// TIA Portal V21 export
FUNCTION "ALARMS" : Void   // FC8, LAD
{ S7_Optimized_Access := 'TRUE' }
// stored: SetENOAutomatically false
   VAR_TEMP   // added for the SCL form of the ladder/FBD networks
      _w1 : Bool;
      _w2 : Bool;
      _w3 : Bool;
      _w4 : Bool;
   END_VAR
BEGIN

REGION Network 1: ERROR
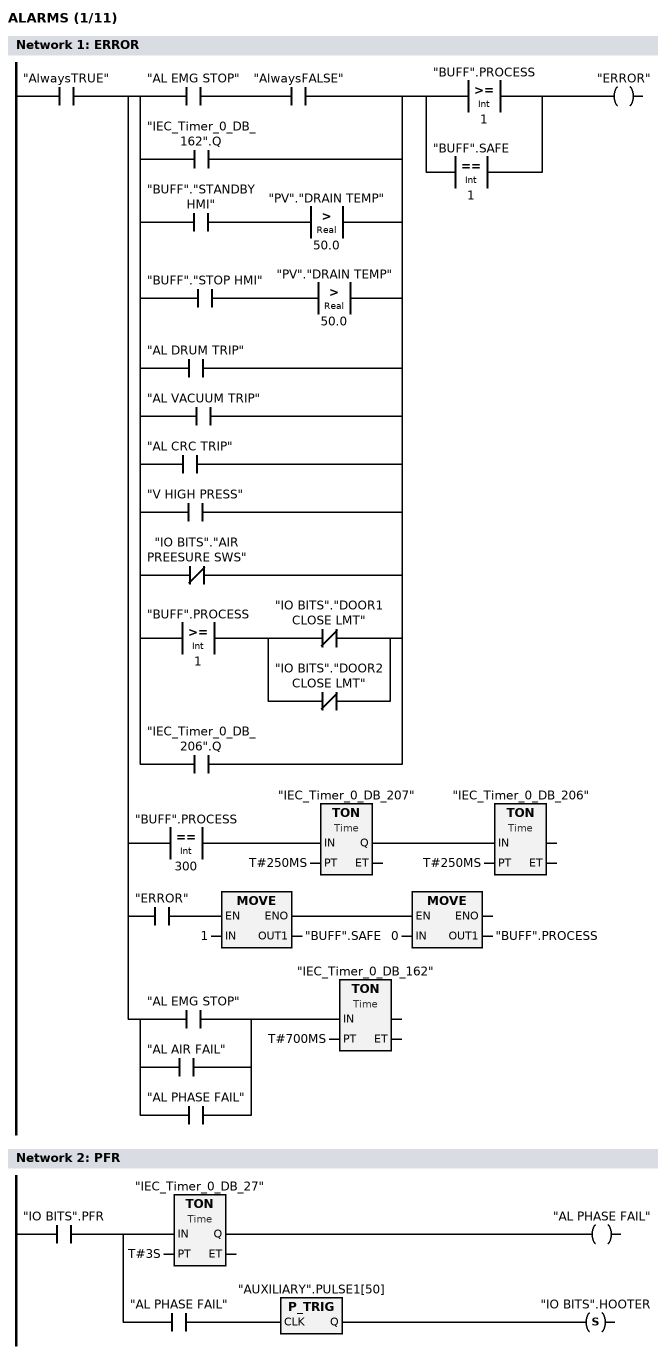
   RUNG wire#powerrail
      Contact( "AlwaysTRUE" )
      wire#w1
      Contact( "AL EMG STOP" )
      Contact( "AlwaysFALSE" )
      wire#w2
      { S7_Templates := "SrcType := Int" } GE_Contact(in1 := "BUFF".PROCESS, in2 := 1)
      wire#w4
      Coil( "ERROR" )
   END_RUNG
   RUNG wire#w1
      Contact( "IEC_Timer_0_DB_162".Q )
   END_RUNG wire#w2
   RUNG wire#w1
      Contact( "BUFF"."STANDBY HMI" )
      { S7_Templates := "SrcType := Real" } GT_Contact(in1 := "PV"."DRAIN TEMP", in2 := 50.0)
   END_RUNG wire#w2
   RUNG wire#w1
      Contact( "BUFF"."STOP HMI" )
      { S7_Templates := "SrcType := Real" } GT_Contact(in1 := "PV"."DRAIN TEMP", in2 := 50.0)
   END_RUNG wire#w2
   RUNG wire#w1
      Contact( "AL DRUM TRIP" )
   END_RUNG wire#w2
   RUNG wire#w1
      Contact( "AL VACUUM TRIP" )
   END_RUNG wire#w2
   RUNG wire#w1
      Contact( "AL CRC TRIP" )
   END_RUNG wire#w2
   RUNG wire#w1
      Contact( "V HIGH PRESS" )
   END_RUNG wire#w2
   RUNG wire#w1
      I_Contact( "IO BITS"."AIR PREESURE SWS" )
   END_RUNG wire#w2
   RUNG wire#w1
      { S7_Templates := "SrcType := Int" } GE_Contact(in1 := "BUFF".PROCESS, in2 := 1)
      wire#w3
      I_Contact( "IO BITS"."DOOR1 CLOSE LMT" )
   END_RUNG wire#w2
   RUNG wire#w3
      I_Contact( "IO BITS"."DOOR2 CLOSE LMT" )
   END_RUNG wire#w2
   RUNG wire#w1
      Contact( "IEC_Timer_0_DB_206".Q )
   END_RUNG wire#w2
   RUNG wire#w2
      { S7_Templates := "SrcType := Int" } EQ_Contact(in1 := "BUFF".SAFE, in2 := 1)
   END_RUNG wire#w4
   RUNG wire#w1
      { S7_Templates := "SrcType := Int" } EQ_Contact(in1 := "BUFF".PROCESS, in2 := 300)
      { S7_Templates := "time_type := Time" } "IEC_Timer_0_DB_207".TON(pt := T#250MS, et =>)
      { S7_Templates := "time_type := Time" } "IEC_Timer_0_DB_206".TON(pt := T#250MS, et =>)
   END_RUNG
   RUNG wire#w1
      Contact( "ERROR" )
      Move(in := 1, out1 => "BUFF".SAFE)
      Move(in := 0, out1 => "BUFF".PROCESS)
   END_RUNG
   RUNG wire#w1
      Contact( "AL EMG STOP" )
      wire#w5
      { S7_Templates := "time_type := Time" } "IEC_Timer_0_DB_162".TON(pt := T#700MS, et =>)
   END_RUNG
   RUNG wire#w1
      Contact( "AL AIR FAIL" )
   END_RUNG wire#w5
   RUNG wire#w1
      Contact( "AL PHASE FAIL" )
   END_RUNG wire#w5
   // the same network as SCL:
   "ERROR" := "AlwaysTRUE" AND (("AL EMG STOP" AND "AlwaysFALSE") OR "IEC_Timer_0_DB_162".Q OR ("BUFF"."STANDBY HMI" AND ("PV"."DRAIN TEMP" > 50.0)) OR ("BUFF"."STOP HMI" AND ("PV"."DRAIN TEMP" > 50.0)) OR "AL DRUM TRIP" OR "AL VACUUM TRIP" OR "AL CRC TRIP" OR "V HIGH PRESS" OR NOT "IO BITS"."AIR PREESURE SWS" OR (("BUFF".PROCESS >= 1) AND (NOT "IO BITS"."DOOR1 CLOSE LMT" OR NOT "IO BITS"."DOOR2 CLOSE LMT")) OR "IEC_Timer_0_DB_206".Q) AND (("BUFF".PROCESS >= 1) OR ("BUFF".SAFE = 1));
   "IEC_Timer_0_DB_207".TON(IN := "AlwaysTRUE" AND ("BUFF".PROCESS = 300), PT := T#250MS);
   "IEC_Timer_0_DB_206".TON(IN := "IEC_Timer_0_DB_207".Q, PT := T#250MS);
   IF "AlwaysTRUE" AND "ERROR" THEN
       "BUFF".SAFE := 1;
       "BUFF".PROCESS := 0;
   END_IF;
   "IEC_Timer_0_DB_162".TON(IN := "AlwaysTRUE" AND ("AL EMG STOP" OR "AL AIR FAIL" OR "AL PHASE FAIL"),
                           PT := T#700MS);
END_REGION

REGION Network 2: PFR
   RUNG wire#powerrail
      Contact( "IO BITS".PFR )
      wire#w1
      { S7_Templates := "time_type := Time" } "IEC_Timer_0_DB_27".TON(pt := T#3S, et =>)
      Coil( "AL PHASE FAIL" )
   END_RUNG
   RUNG wire#w1
      Contact( "AL PHASE FAIL" )
      P_Trig( "AUXILIARY".PULSE1[50] )
      S_Coil( "IO BITS".HOOTER )
   END_RUNG
   // the same network as SCL:
   "IEC_Timer_0_DB_27".TON(IN := "IO BITS".PFR, PT := T#3S);
   "AL PHASE FAIL" := "IEC_Timer_0_DB_27".Q;
   #_w1 := "IO BITS".PFR AND "AL PHASE FAIL";
   #_w2 := #_w1 AND NOT "AUXILIARY".PULSE1[50];   // rising edge
   "AUXILIARY".PULSE1[50] := #_w1;
   IF #_w2 THEN "IO BITS".HOOTER := TRUE; END_IF;
END_REGION

REGION Network 3: EMG
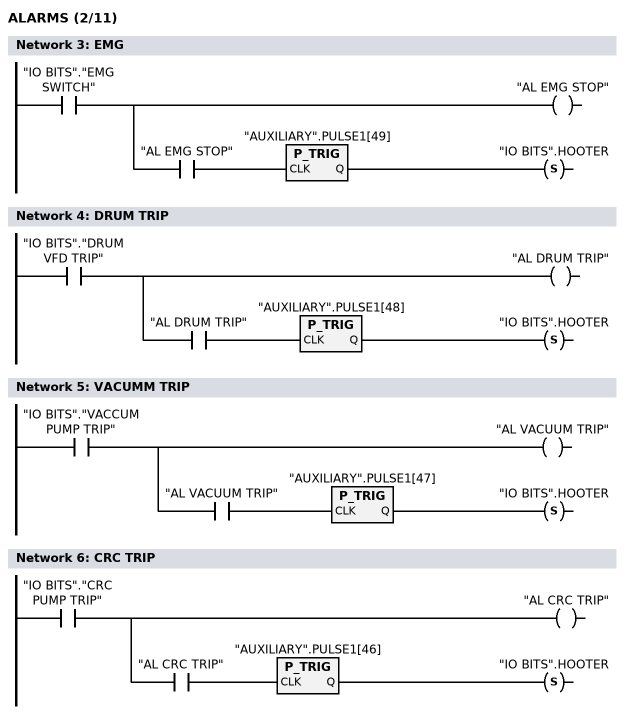
   RUNG wire#powerrail
      Contact( "IO BITS"."EMG SWITCH" )
      wire#w1
      Coil( "AL EMG STOP" )
   END_RUNG
   RUNG wire#w1
      Contact( "AL EMG STOP" )
      P_Trig( "AUXILIARY".PULSE1[49] )
      S_Coil( "IO BITS".HOOTER )
   END_RUNG
   // the same network as SCL:
   "AL EMG STOP" := "IO BITS"."EMG SWITCH";
   #_w1 := "IO BITS"."EMG SWITCH" AND "AL EMG STOP";
   #_w2 := #_w1 AND NOT "AUXILIARY".PULSE1[49];   // rising edge
   "AUXILIARY".PULSE1[49] := #_w1;
   IF #_w2 THEN "IO BITS".HOOTER := TRUE; END_IF;
END_REGION

REGION Network 4: DRUM TRIP
   RUNG wire#powerrail
      Contact( "IO BITS"."DRUM VFD TRIP" )
      wire#w1
      Coil( "AL DRUM TRIP" )
   END_RUNG
   RUNG wire#w1
      Contact( "AL DRUM TRIP" )
      P_Trig( "AUXILIARY".PULSE1[48] )
      S_Coil( "IO BITS".HOOTER )
   END_RUNG
   // the same network as SCL:
   "AL DRUM TRIP" := "IO BITS"."DRUM VFD TRIP";
   #_w1 := "IO BITS"."DRUM VFD TRIP" AND "AL DRUM TRIP";
   #_w2 := #_w1 AND NOT "AUXILIARY".PULSE1[48];   // rising edge
   "AUXILIARY".PULSE1[48] := #_w1;
   IF #_w2 THEN "IO BITS".HOOTER := TRUE; END_IF;
END_REGION

REGION Network 5: VACUMM TRIP
   RUNG wire#powerrail
      Contact( "IO BITS"."VACCUM PUMP TRIP" )
      wire#w1
      Coil( "AL VACUUM TRIP" )
   END_RUNG
   RUNG wire#w1
      Contact( "AL VACUUM TRIP" )
      P_Trig( "AUXILIARY".PULSE1[47] )
      S_Coil( "IO BITS".HOOTER )
   END_RUNG
   // the same network as SCL:
   "AL VACUUM TRIP" := "IO BITS"."VACCUM PUMP TRIP";
   #_w1 := "IO BITS"."VACCUM PUMP TRIP" AND "AL VACUUM TRIP";
   #_w2 := #_w1 AND NOT "AUXILIARY".PULSE1[47];   // rising edge
   "AUXILIARY".PULSE1[47] := #_w1;
   IF #_w2 THEN "IO BITS".HOOTER := TRUE; END_IF;
END_REGION

REGION Network 6: CRC TRIP
   RUNG wire#powerrail
      Contact( "IO BITS"."CRC PUMP TRIP" )
      wire#w1
      Coil( "AL CRC TRIP" )
   END_RUNG
   RUNG wire#w1
      Contact( "AL CRC TRIP" )
      P_Trig( "AUXILIARY".PULSE1[46] )
      S_Coil( "IO BITS".HOOTER )
   END_RUNG
   // the same network as SCL:
   "AL CRC TRIP" := "IO BITS"."CRC PUMP TRIP";
   #_w1 := "IO BITS"."CRC PUMP TRIP" AND "AL CRC TRIP";
   #_w2 := #_w1 AND NOT "AUXILIARY".PULSE1[46];   // rising edge
   "AUXILIARY".PULSE1[46] := #_w1;
   IF #_w2 THEN "IO BITS".HOOTER := TRUE; END_IF;
END_REGION

REGION Network 7: PROCESS START AND OVER
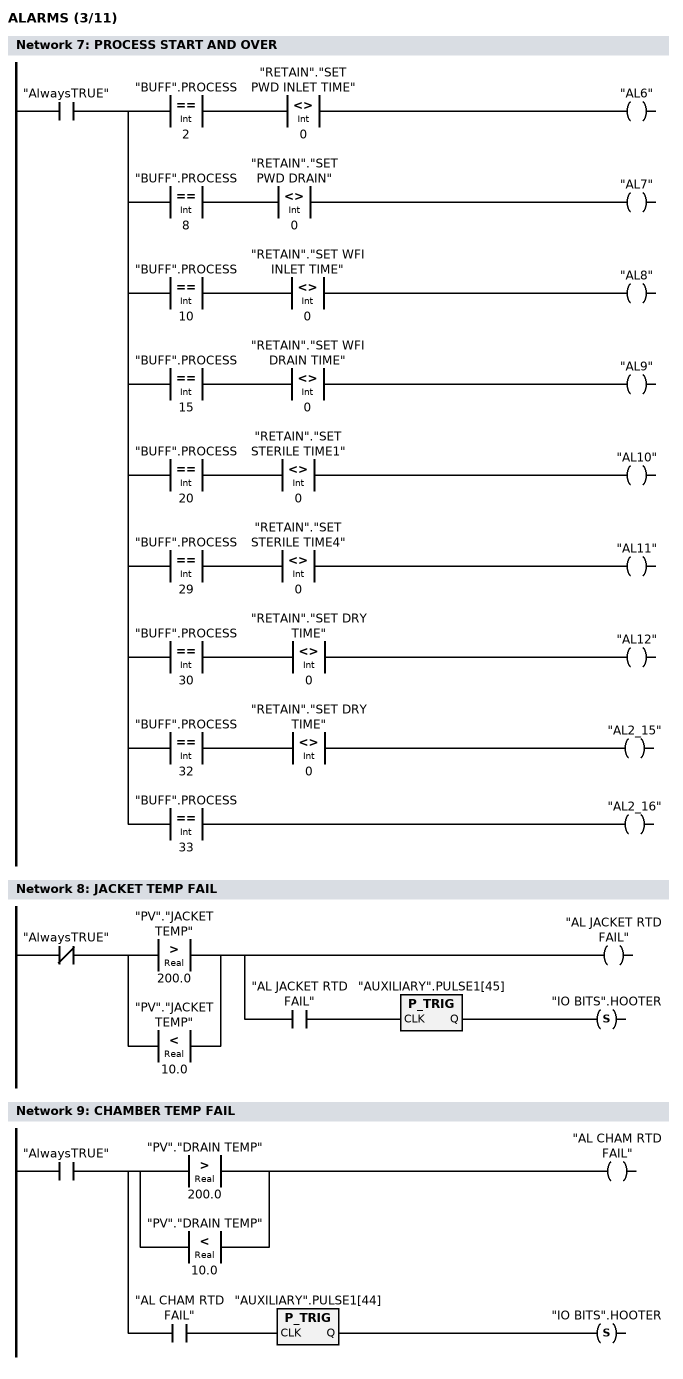
   RUNG wire#powerrail
      Contact( "AlwaysTRUE" )
      wire#w1
      { S7_Templates := "SrcType := Int" } EQ_Contact(in1 := "BUFF".PROCESS, in2 := 2)
      { S7_Templates := "SrcType := Int" } NE_Contact(in1 := "RETAIN"."SET PWD INLET TIME", in2 := 0)
      Coil( "AL6" )
   END_RUNG
   RUNG wire#w1
      { S7_Templates := "SrcType := Int" } EQ_Contact(in1 := "BUFF".PROCESS, in2 := 8)
      { S7_Templates := "SrcType := Int" } NE_Contact(in1 := "RETAIN"."SET PWD DRAIN", in2 := 0)
      Coil( "AL7" )
   END_RUNG
   RUNG wire#w1
      { S7_Templates := "SrcType := Int" } EQ_Contact(in1 := "BUFF".PROCESS, in2 := 10)
      { S7_Templates := "SrcType := Int" } NE_Contact(in1 := "RETAIN"."SET WFI INLET TIME", in2 := 0)
      Coil( "AL8" )
   END_RUNG
   RUNG wire#w1
      { S7_Templates := "SrcType := Int" } EQ_Contact(in1 := "BUFF".PROCESS, in2 := 15)
      { S7_Templates := "SrcType := Int" } NE_Contact(in1 := "RETAIN"."SET WFI DRAIN TIME", in2 := 0)
      Coil( "AL9" )
   END_RUNG
   RUNG wire#w1
      { S7_Templates := "SrcType := Int" } EQ_Contact(in1 := "BUFF".PROCESS, in2 := 20)
      { S7_Templates := "SrcType := Int" } NE_Contact(in1 := "RETAIN"."SET STERILE TIME1", in2 := 0)
      Coil( "AL10" )
   END_RUNG
   RUNG wire#w1
      { S7_Templates := "SrcType := Int" } EQ_Contact(in1 := "BUFF".PROCESS, in2 := 29)
      { S7_Templates := "SrcType := Int" } NE_Contact(in1 := "RETAIN"."SET STERILE TIME4", in2 := 0)
      Coil( "AL11" )
   END_RUNG
   RUNG wire#w1
      { S7_Templates := "SrcType := Int" } EQ_Contact(in1 := "BUFF".PROCESS, in2 := 30)
      { S7_Templates := "SrcType := Int" } NE_Contact(in1 := "RETAIN"."SET DRY TIME", in2 := 0)
      Coil( "AL12" )
   END_RUNG
   RUNG wire#w1
      { S7_Templates := "SrcType := Int" } EQ_Contact(in1 := "BUFF".PROCESS, in2 := 32)
      { S7_Templates := "SrcType := Int" } NE_Contact(in1 := "RETAIN"."SET DRY TIME", in2 := 0)
      Coil( "AL2_15" )
   END_RUNG
   RUNG wire#w1
      { S7_Templates := "SrcType := Int" } EQ_Contact(in1 := "BUFF".PROCESS, in2 := 33)
      Coil( "AL2_16" )
   END_RUNG
   // the same network as SCL:
   "AL6" := "AlwaysTRUE" AND ("BUFF".PROCESS = 2) AND ("RETAIN"."SET PWD INLET TIME" <> 0);
   "AL7" := "AlwaysTRUE" AND ("BUFF".PROCESS = 8) AND ("RETAIN"."SET PWD DRAIN" <> 0);
   "AL8" := "AlwaysTRUE" AND ("BUFF".PROCESS = 10) AND ("RETAIN"."SET WFI INLET TIME" <> 0);
   "AL9" := "AlwaysTRUE" AND ("BUFF".PROCESS = 15) AND ("RETAIN"."SET WFI DRAIN TIME" <> 0);
   "AL10" := "AlwaysTRUE" AND ("BUFF".PROCESS = 20) AND ("RETAIN"."SET STERILE TIME1" <> 0);
   "AL11" := "AlwaysTRUE" AND ("BUFF".PROCESS = 29) AND ("RETAIN"."SET STERILE TIME4" <> 0);
   "AL12" := "AlwaysTRUE" AND ("BUFF".PROCESS = 30) AND ("RETAIN"."SET DRY TIME" <> 0);
   "AL2_15" := "AlwaysTRUE" AND ("BUFF".PROCESS = 32) AND ("RETAIN"."SET DRY TIME" <> 0);
   "AL2_16" := "AlwaysTRUE" AND ("BUFF".PROCESS = 33);
END_REGION

REGION Network 8: JACKET TEMP FAIL
   RUNG wire#powerrail
      I_Contact( "AlwaysTRUE" )
      wire#w1
      { S7_Templates := "SrcType := Real" } GT_Contact(in1 := "PV"."JACKET TEMP", in2 := 200.0)
      wire#w2
      Coil( "AL JACKET RTD FAIL" )
   END_RUNG
   RUNG wire#w1
      { S7_Templates := "SrcType := Real" } LT_Contact(in1 := "PV"."JACKET TEMP", in2 := 10.0)
   END_RUNG wire#w2
   RUNG wire#w2
      Contact( "AL JACKET RTD FAIL" )
      P_Trig( "AUXILIARY".PULSE1[45] )
      S_Coil( "IO BITS".HOOTER )
   END_RUNG
   // the same network as SCL:
   "AL JACKET RTD FAIL" := NOT "AlwaysTRUE" AND (("PV"."JACKET TEMP" > 200.0) OR ("PV"."JACKET TEMP" < 10.0));
   #_w1 := "AL JACKET RTD FAIL" AND "AL JACKET RTD FAIL";
   #_w2 := #_w1 AND NOT "AUXILIARY".PULSE1[45];   // rising edge
   "AUXILIARY".PULSE1[45] := #_w1;
   IF #_w2 THEN "IO BITS".HOOTER := TRUE; END_IF;
END_REGION

REGION Network 9: CHAMBER TEMP FAIL
   RUNG wire#powerrail
      Contact( "AlwaysTRUE" )
      wire#w1
      { S7_Templates := "SrcType := Real" } GT_Contact(in1 := "PV"."DRAIN TEMP", in2 := 200.0)
      wire#w2
      Coil( "AL CHAM RTD FAIL" )
   END_RUNG
   RUNG wire#w1
      { S7_Templates := "SrcType := Real" } LT_Contact(in1 := "PV"."DRAIN TEMP", in2 := 10.0)
   END_RUNG wire#w2
   RUNG wire#w1
      Contact( "AL CHAM RTD FAIL" )
      P_Trig( "AUXILIARY".PULSE1[44] )
      S_Coil( "IO BITS".HOOTER )
   END_RUNG
   // the same network as SCL:
   "AL CHAM RTD FAIL" := "AlwaysTRUE" AND (("PV"."DRAIN TEMP" > 200.0) OR ("PV"."DRAIN TEMP" < 10.0));
   #_w1 := "AlwaysTRUE" AND "AL CHAM RTD FAIL";
   #_w2 := #_w1 AND NOT "AUXILIARY".PULSE1[44];   // rising edge
   "AUXILIARY".PULSE1[44] := #_w1;
   IF #_w2 THEN "IO BITS".HOOTER := TRUE; END_IF;
END_REGION

REGION Network 10: AIR FAIL
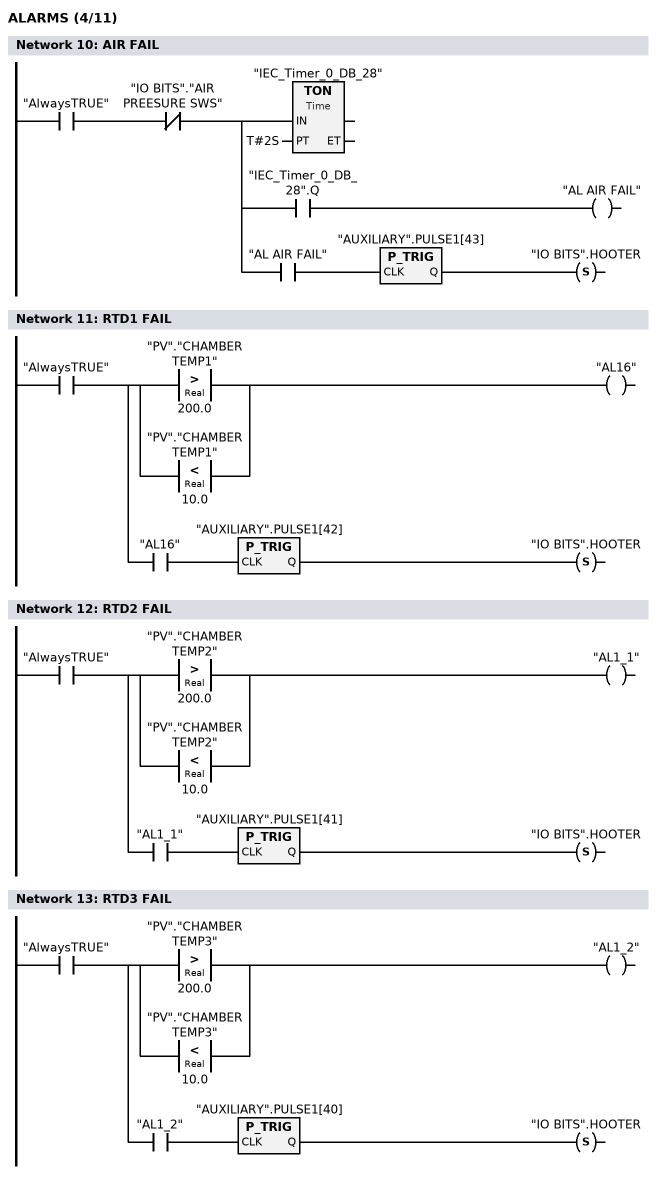
   RUNG wire#powerrail
      Contact( "AlwaysTRUE" )
      I_Contact( "IO BITS"."AIR PREESURE SWS" )
      wire#w1
      { S7_Templates := "time_type := Time" } "IEC_Timer_0_DB_28".TON(pt := T#2S, et =>)
   END_RUNG
   RUNG wire#w1
      Contact( "IEC_Timer_0_DB_28".Q )
      Coil( "AL AIR FAIL" )
   END_RUNG
   RUNG wire#w1
      Contact( "AL AIR FAIL" )
      P_Trig( "AUXILIARY".PULSE1[43] )
      S_Coil( "IO BITS".HOOTER )
   END_RUNG
   // the same network as SCL:
   #_w1 := "AlwaysTRUE" AND NOT "IO BITS"."AIR PREESURE SWS";
   "IEC_Timer_0_DB_28".TON(IN := #_w1, PT := T#2S);
   "AL AIR FAIL" := #_w1 AND "IEC_Timer_0_DB_28".Q;
   #_w2 := #_w1 AND "AL AIR FAIL";
   #_w3 := #_w2 AND NOT "AUXILIARY".PULSE1[43];   // rising edge
   "AUXILIARY".PULSE1[43] := #_w2;
   IF #_w3 THEN "IO BITS".HOOTER := TRUE; END_IF;
END_REGION

REGION Network 11: RTD1 FAIL
   RUNG wire#powerrail
      Contact( "AlwaysTRUE" )
      wire#w1
      { S7_Templates := "SrcType := Real" } GT_Contact(in1 := "PV"."CHAMBER TEMP1", in2 := 200.0)
      wire#w2
      Coil( "AL16" )
   END_RUNG
   RUNG wire#w1
      { S7_Templates := "SrcType := Real" } LT_Contact(in1 := "PV"."CHAMBER TEMP1", in2 := 10.0)
   END_RUNG wire#w2
   RUNG wire#w1
      Contact( "AL16" )
      P_Trig( "AUXILIARY".PULSE1[42] )
      S_Coil( "IO BITS".HOOTER )
   END_RUNG
   // the same network as SCL:
   "AL16" := "AlwaysTRUE" AND (("PV"."CHAMBER TEMP1" > 200.0) OR ("PV"."CHAMBER TEMP1" < 10.0));
   #_w1 := "AlwaysTRUE" AND "AL16";
   #_w2 := #_w1 AND NOT "AUXILIARY".PULSE1[42];   // rising edge
   "AUXILIARY".PULSE1[42] := #_w1;
   IF #_w2 THEN "IO BITS".HOOTER := TRUE; END_IF;
END_REGION

REGION Network 12: RTD2 FAIL
   RUNG wire#powerrail
      Contact( "AlwaysTRUE" )
      wire#w1
      { S7_Templates := "SrcType := Real" } GT_Contact(in1 := "PV"."CHAMBER TEMP2", in2 := 200.0)
      wire#w2
      Coil( "AL1_1" )
   END_RUNG
   RUNG wire#w1
      { S7_Templates := "SrcType := Real" } LT_Contact(in1 := "PV"."CHAMBER TEMP2", in2 := 10.0)
   END_RUNG wire#w2
   RUNG wire#w1
      Contact( "AL1_1" )
      P_Trig( "AUXILIARY".PULSE1[41] )
      S_Coil( "IO BITS".HOOTER )
   END_RUNG
   // the same network as SCL:
   "AL1_1" := "AlwaysTRUE" AND (("PV"."CHAMBER TEMP2" > 200.0) OR ("PV"."CHAMBER TEMP2" < 10.0));
   #_w1 := "AlwaysTRUE" AND "AL1_1";
   #_w2 := #_w1 AND NOT "AUXILIARY".PULSE1[41];   // rising edge
   "AUXILIARY".PULSE1[41] := #_w1;
   IF #_w2 THEN "IO BITS".HOOTER := TRUE; END_IF;
END_REGION

REGION Network 13: RTD3 FAIL
   RUNG wire#powerrail
      Contact( "AlwaysTRUE" )
      wire#w1
      { S7_Templates := "SrcType := Real" } GT_Contact(in1 := "PV"."CHAMBER TEMP3", in2 := 200.0)
      wire#w2
      Coil( "AL1_2" )
   END_RUNG
   RUNG wire#w1
      { S7_Templates := "SrcType := Real" } LT_Contact(in1 := "PV"."CHAMBER TEMP3", in2 := 10.0)
   END_RUNG wire#w2
   RUNG wire#w1
      Contact( "AL1_2" )
      P_Trig( "AUXILIARY".PULSE1[40] )
      S_Coil( "IO BITS".HOOTER )
   END_RUNG
   // the same network as SCL:
   "AL1_2" := "AlwaysTRUE" AND (("PV"."CHAMBER TEMP3" > 200.0) OR ("PV"."CHAMBER TEMP3" < 10.0));
   #_w1 := "AlwaysTRUE" AND "AL1_2";
   #_w2 := #_w1 AND NOT "AUXILIARY".PULSE1[40];   // rising edge
   "AUXILIARY".PULSE1[40] := #_w1;
   IF #_w2 THEN "IO BITS".HOOTER := TRUE; END_IF;
END_REGION

REGION Network 14: RTD4 FAIL
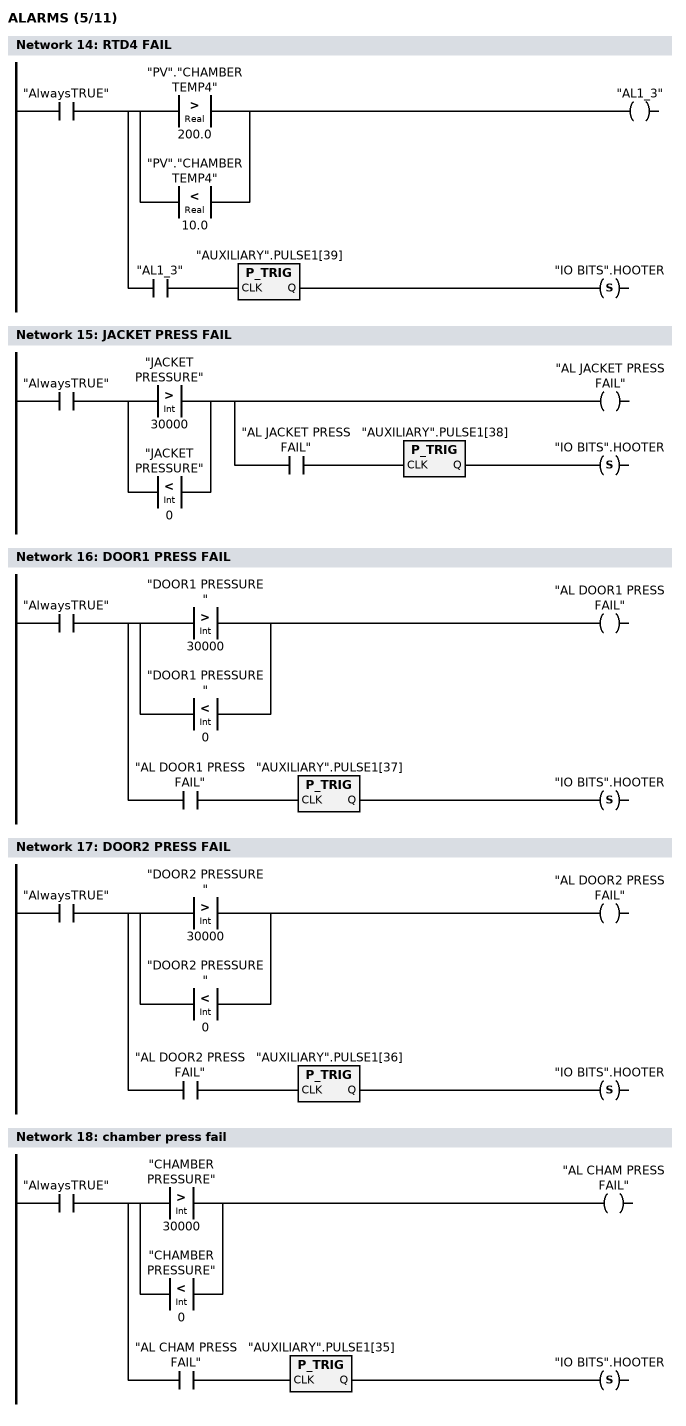
   RUNG wire#powerrail
      Contact( "AlwaysTRUE" )
      wire#w1
      { S7_Templates := "SrcType := Real" } GT_Contact(in1 := "PV"."CHAMBER TEMP4", in2 := 200.0)
      wire#w2
      Coil( "AL1_3" )
   END_RUNG
   RUNG wire#w1
      { S7_Templates := "SrcType := Real" } LT_Contact(in1 := "PV"."CHAMBER TEMP4", in2 := 10.0)
   END_RUNG wire#w2
   RUNG wire#w1
      Contact( "AL1_3" )
      P_Trig( "AUXILIARY".PULSE1[39] )
      S_Coil( "IO BITS".HOOTER )
   END_RUNG
   // the same network as SCL:
   "AL1_3" := "AlwaysTRUE" AND (("PV"."CHAMBER TEMP4" > 200.0) OR ("PV"."CHAMBER TEMP4" < 10.0));
   #_w1 := "AlwaysTRUE" AND "AL1_3";
   #_w2 := #_w1 AND NOT "AUXILIARY".PULSE1[39];   // rising edge
   "AUXILIARY".PULSE1[39] := #_w1;
   IF #_w2 THEN "IO BITS".HOOTER := TRUE; END_IF;
END_REGION

REGION Network 15: JACKET PRESS FAIL
   RUNG wire#powerrail
      Contact( "AlwaysTRUE" )
      wire#w1
      { S7_Templates := "SrcType := Int" } GT_Contact(in1 := "JACKET PRESSURE", in2 := 30000)
      wire#w2
      Coil( "AL JACKET PRESS FAIL" )
   END_RUNG
   RUNG wire#w1
      { S7_Templates := "SrcType := Int" } LT_Contact(in1 := "JACKET PRESSURE", in2 := 0)
   END_RUNG wire#w2
   RUNG wire#w2
      Contact( "AL JACKET PRESS FAIL" )
      P_Trig( "AUXILIARY".PULSE1[38] )
      S_Coil( "IO BITS".HOOTER )
   END_RUNG
   // the same network as SCL:
   "AL JACKET PRESS FAIL" := "AlwaysTRUE" AND (("JACKET PRESSURE" > 30000) OR ("JACKET PRESSURE" < 0));
   #_w1 := "AL JACKET PRESS FAIL" AND "AL JACKET PRESS FAIL";
   #_w2 := #_w1 AND NOT "AUXILIARY".PULSE1[38];   // rising edge
   "AUXILIARY".PULSE1[38] := #_w1;
   IF #_w2 THEN "IO BITS".HOOTER := TRUE; END_IF;
END_REGION

REGION Network 16: DOOR1 PRESS FAIL
   RUNG wire#powerrail
      Contact( "AlwaysTRUE" )
      wire#w1
      { S7_Templates := "SrcType := Int" } GT_Contact(in1 := "DOOR1 PRESSURE", in2 := 30000)
      wire#w2
      Coil( "AL DOOR1 PRESS FAIL" )
   END_RUNG
   RUNG wire#w1
      { S7_Templates := "SrcType := Int" } LT_Contact(in1 := "DOOR1 PRESSURE", in2 := 0)
   END_RUNG wire#w2
   RUNG wire#w1
      Contact( "AL DOOR1 PRESS FAIL" )
      P_Trig( "AUXILIARY".PULSE1[37] )
      S_Coil( "IO BITS".HOOTER )
   END_RUNG
   // the same network as SCL:
   "AL DOOR1 PRESS FAIL" := "AlwaysTRUE" AND (("DOOR1 PRESSURE" > 30000) OR ("DOOR1 PRESSURE" < 0));
   #_w1 := "AlwaysTRUE" AND "AL DOOR1 PRESS FAIL";
   #_w2 := #_w1 AND NOT "AUXILIARY".PULSE1[37];   // rising edge
   "AUXILIARY".PULSE1[37] := #_w1;
   IF #_w2 THEN "IO BITS".HOOTER := TRUE; END_IF;
END_REGION

REGION Network 17: DOOR2 PRESS FAIL
   RUNG wire#powerrail
      Contact( "AlwaysTRUE" )
      wire#w1
      { S7_Templates := "SrcType := Int" } GT_Contact(in1 := "DOOR2 PRESSURE", in2 := 30000)
      wire#w2
      Coil( "AL DOOR2 PRESS FAIL" )
   END_RUNG
   RUNG wire#w1
      { S7_Templates := "SrcType := Int" } LT_Contact(in1 := "DOOR2 PRESSURE", in2 := 0)
   END_RUNG wire#w2
   RUNG wire#w1
      Contact( "AL DOOR2 PRESS FAIL" )
      P_Trig( "AUXILIARY".PULSE1[36] )
      S_Coil( "IO BITS".HOOTER )
   END_RUNG
   // the same network as SCL:
   "AL DOOR2 PRESS FAIL" := "AlwaysTRUE" AND (("DOOR2 PRESSURE" > 30000) OR ("DOOR2 PRESSURE" < 0));
   #_w1 := "AlwaysTRUE" AND "AL DOOR2 PRESS FAIL";
   #_w2 := #_w1 AND NOT "AUXILIARY".PULSE1[36];   // rising edge
   "AUXILIARY".PULSE1[36] := #_w1;
   IF #_w2 THEN "IO BITS".HOOTER := TRUE; END_IF;
END_REGION

REGION Network 18: chamber press fail
   RUNG wire#powerrail
      Contact( "AlwaysTRUE" )
      wire#w1
      { S7_Templates := "SrcType := Int" } GT_Contact(in1 := "CHAMBER PRESSURE", in2 := 30000)
      wire#w2
      Coil( "AL CHAM PRESS FAIL" )
   END_RUNG
   RUNG wire#w1
      { S7_Templates := "SrcType := Int" } LT_Contact(in1 := "CHAMBER PRESSURE", in2 := 0)
   END_RUNG wire#w2
   RUNG wire#w1
      Contact( "AL CHAM PRESS FAIL" )
      P_Trig( "AUXILIARY".PULSE1[35] )
      S_Coil( "IO BITS".HOOTER )
   END_RUNG
   // the same network as SCL:
   "AL CHAM PRESS FAIL" := "AlwaysTRUE" AND (("CHAMBER PRESSURE" > 30000) OR ("CHAMBER PRESSURE" < 0));
   #_w1 := "AlwaysTRUE" AND "AL CHAM PRESS FAIL";
   #_w2 := #_w1 AND NOT "AUXILIARY".PULSE1[35];   // rising edge
   "AUXILIARY".PULSE1[35] := #_w1;
   IF #_w2 THEN "IO BITS".HOOTER := TRUE; END_IF;
END_REGION

REGION Network 19: door limit fail
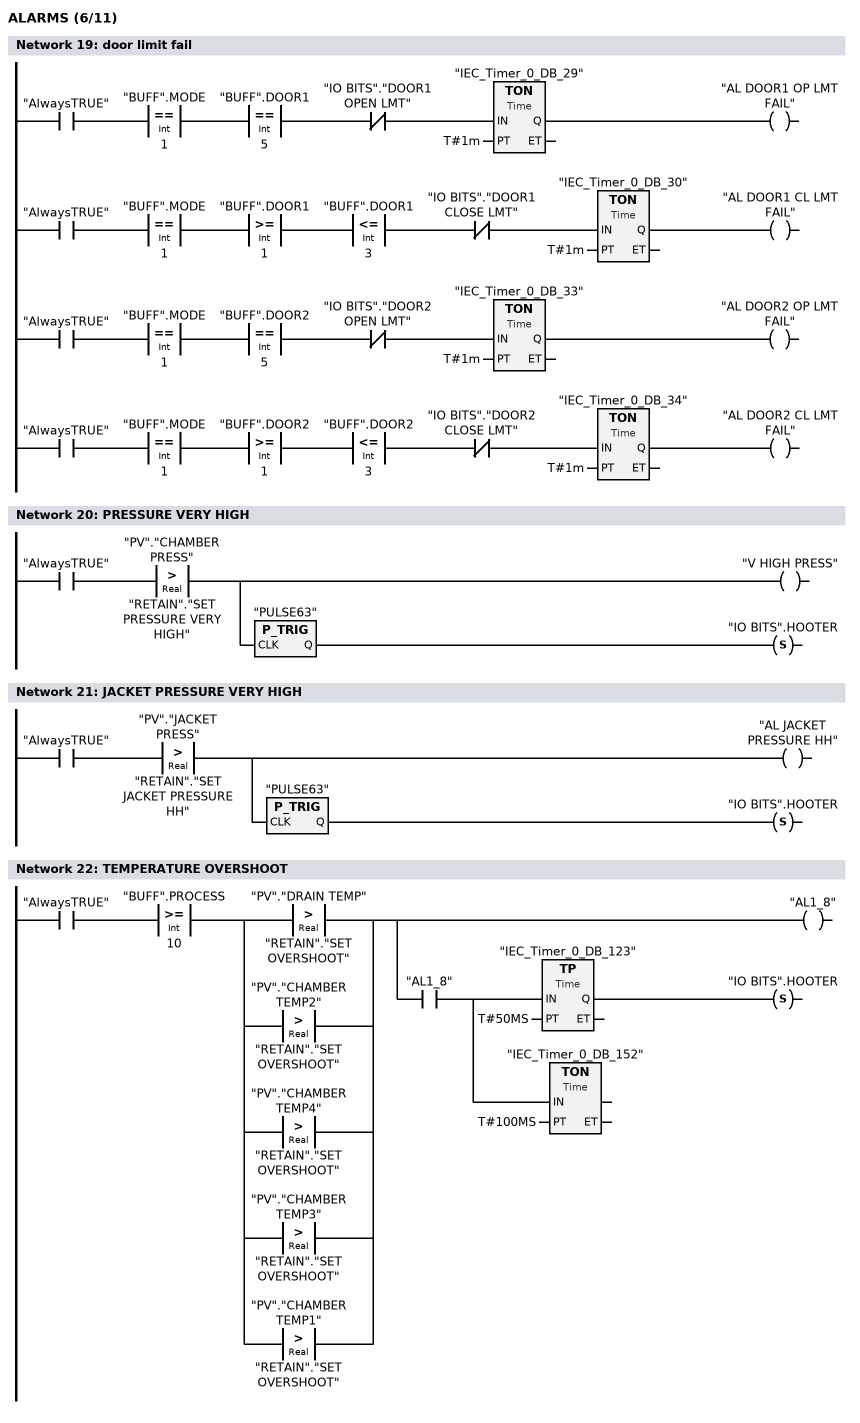
   RUNG wire#powerrail
      Contact( "AlwaysTRUE" )
      { S7_Templates := "SrcType := Int" } EQ_Contact(in1 := "BUFF".MODE, in2 := 1)
      { S7_Templates := "SrcType := Int" } EQ_Contact(in1 := "BUFF".DOOR1, in2 := 5)
      I_Contact( "IO BITS"."DOOR1 OPEN LMT" )
      { S7_Templates := "time_type := Time" } "IEC_Timer_0_DB_29".TON(pt := T#1m, et =>)
      Coil( "AL DOOR1 OP LMT FAIL" )
   END_RUNG
   RUNG wire#powerrail
      Contact( "AlwaysTRUE" )
      { S7_Templates := "SrcType := Int" } EQ_Contact(in1 := "BUFF".MODE, in2 := 1)
      { S7_Templates := "SrcType := Int" } GE_Contact(in1 := "BUFF".DOOR1, in2 := 1)
      { S7_Templates := "SrcType := Int" } LE_Contact(in1 := "BUFF".DOOR1, in2 := 3)
      I_Contact( "IO BITS"."DOOR1 CLOSE LMT" )
      { S7_Templates := "time_type := Time" } "IEC_Timer_0_DB_30".TON(pt := T#1m, et =>)
      Coil( "AL DOOR1 CL LMT FAIL" )
   END_RUNG
   RUNG wire#powerrail
      Contact( "AlwaysTRUE" )
      { S7_Templates := "SrcType := Int" } EQ_Contact(in1 := "BUFF".MODE, in2 := 1)
      { S7_Templates := "SrcType := Int" } EQ_Contact(in1 := "BUFF".DOOR2, in2 := 5)
      I_Contact( "IO BITS"."DOOR2 OPEN LMT" )
      { S7_Templates := "time_type := Time" } "IEC_Timer_0_DB_33".TON(pt := T#1m, et =>)
      Coil( "AL DOOR2 OP LMT FAIL" )
   END_RUNG
   RUNG wire#powerrail
      Contact( "AlwaysTRUE" )
      { S7_Templates := "SrcType := Int" } EQ_Contact(in1 := "BUFF".MODE, in2 := 1)
      { S7_Templates := "SrcType := Int" } GE_Contact(in1 := "BUFF".DOOR2, in2 := 1)
      { S7_Templates := "SrcType := Int" } LE_Contact(in1 := "BUFF".DOOR2, in2 := 3)
      I_Contact( "IO BITS"."DOOR2 CLOSE LMT" )
      { S7_Templates := "time_type := Time" } "IEC_Timer_0_DB_34".TON(pt := T#1m, et =>)
      Coil( "AL DOOR2 CL LMT FAIL" )
   END_RUNG
   // the same network as SCL:
   "IEC_Timer_0_DB_29".TON(IN := "AlwaysTRUE" AND ("BUFF".MODE = 1) AND ("BUFF".DOOR1 = 5) AND NOT "IO BITS"."DOOR1 OPEN LMT",
                           PT := T#1m);
   "AL DOOR1 OP LMT FAIL" := "IEC_Timer_0_DB_29".Q;
   "IEC_Timer_0_DB_30".TON(IN := "AlwaysTRUE" AND ("BUFF".MODE = 1) AND ("BUFF".DOOR1 >= 1) AND ("BUFF".DOOR1 <= 3) AND NOT "IO BITS"."DOOR1 CLOSE LMT",
                           PT := T#1m);
   "AL DOOR1 CL LMT FAIL" := "IEC_Timer_0_DB_30".Q;
   "IEC_Timer_0_DB_33".TON(IN := "AlwaysTRUE" AND ("BUFF".MODE = 1) AND ("BUFF".DOOR2 = 5) AND NOT "IO BITS"."DOOR2 OPEN LMT",
                           PT := T#1m);
   "AL DOOR2 OP LMT FAIL" := "IEC_Timer_0_DB_33".Q;
   "IEC_Timer_0_DB_34".TON(IN := "AlwaysTRUE" AND ("BUFF".MODE = 1) AND ("BUFF".DOOR2 >= 1) AND ("BUFF".DOOR2 <= 3) AND NOT "IO BITS"."DOOR2 CLOSE LMT",
                           PT := T#1m);
   "AL DOOR2 CL LMT FAIL" := "IEC_Timer_0_DB_34".Q;
END_REGION

REGION Network 20: PRESSURE VERY HIGH
   RUNG wire#powerrail
      Contact( "AlwaysTRUE" )
      { S7_Templates := "SrcType := Real" } GT_Contact(in1 := "PV"."CHAMBER PRESS", in2 := "RETAIN"."SET PRESSURE VERY HIGH")
      wire#w1
      Coil( "V HIGH PRESS" )
   END_RUNG
   RUNG wire#w1
      P_Trig( "PULSE63" )
      S_Coil( "IO BITS".HOOTER )
   END_RUNG
   // the same network as SCL:
   "V HIGH PRESS" := "AlwaysTRUE" AND ("PV"."CHAMBER PRESS" > "RETAIN"."SET PRESSURE VERY HIGH");
   #_w1 := "V HIGH PRESS" AND NOT "PULSE63";   // rising edge
   "PULSE63" := "V HIGH PRESS";
   IF #_w1 THEN "IO BITS".HOOTER := TRUE; END_IF;
END_REGION

REGION Network 21: JACKET PRESSURE VERY HIGH
   RUNG wire#powerrail
      Contact( "AlwaysTRUE" )
      { S7_Templates := "SrcType := Real" } GT_Contact(in1 := "PV"."JACKET PRESS", in2 := "RETAIN"."SET JACKET PRESSURE HH")
      wire#w1
      Coil( "AL JACKET PRESSURE HH" )
   END_RUNG
   RUNG wire#w1
      P_Trig( "PULSE63" )
      S_Coil( "IO BITS".HOOTER )
   END_RUNG
   // the same network as SCL:
   "AL JACKET PRESSURE HH" := "AlwaysTRUE" AND ("PV"."JACKET PRESS" > "RETAIN"."SET JACKET PRESSURE HH");
   #_w1 := "AL JACKET PRESSURE HH" AND NOT "PULSE63";   // rising edge
   "PULSE63" := "AL JACKET PRESSURE HH";
   IF #_w1 THEN "IO BITS".HOOTER := TRUE; END_IF;
END_REGION

REGION Network 22: TEMPERATURE OVERSHOOT
   RUNG wire#powerrail
      Contact( "AlwaysTRUE" )
      { S7_Templates := "SrcType := Int" } GE_Contact(in1 := "BUFF".PROCESS, in2 := 10)
      wire#w1
      { S7_Templates := "SrcType := Real" } GT_Contact(in1 := "PV"."DRAIN TEMP", in2 := "RETAIN"."SET OVERSHOOT")
      wire#w2
      Coil( "AL1_8" )
   END_RUNG
   RUNG wire#w1
      { S7_Templates := "SrcType := Real" } GT_Contact(in1 := "PV"."CHAMBER TEMP2", in2 := "RETAIN"."SET OVERSHOOT")
   END_RUNG wire#w2
   RUNG wire#w1
      { S7_Templates := "SrcType := Real" } GT_Contact(in1 := "PV"."CHAMBER TEMP4", in2 := "RETAIN"."SET OVERSHOOT")
   END_RUNG wire#w2
   RUNG wire#w1
      { S7_Templates := "SrcType := Real" } GT_Contact(in1 := "PV"."CHAMBER TEMP3", in2 := "RETAIN"."SET OVERSHOOT")
   END_RUNG wire#w2
   RUNG wire#w1
      { S7_Templates := "SrcType := Real" } GT_Contact(in1 := "PV"."CHAMBER TEMP1", in2 := "RETAIN"."SET OVERSHOOT")
   END_RUNG wire#w2
   RUNG wire#w2
      Contact( "AL1_8" )
      wire#w3
      { S7_Templates := "time_type := Time" } "IEC_Timer_0_DB_123".TP(pt := T#50MS, et =>)
      S_Coil( "IO BITS".HOOTER )
   END_RUNG
   RUNG wire#w3
      { S7_Templates := "time_type := Time" } "IEC_Timer_0_DB_152".TON(pt := T#100MS, et =>)
   END_RUNG
   // the same network as SCL:
   "AL1_8" := "AlwaysTRUE" AND ("BUFF".PROCESS >= 10) AND (("PV"."DRAIN TEMP" > "RETAIN"."SET OVERSHOOT") OR ("PV"."CHAMBER TEMP2" > "RETAIN"."SET OVERSHOOT") OR ("PV"."CHAMBER TEMP4" > "RETAIN"."SET OVERSHOOT") OR ("PV"."CHAMBER TEMP3" > "RETAIN"."SET OVERSHOOT") OR ("PV"."CHAMBER TEMP1" > "RETAIN"."SET OVERSHOOT"));
   #_w1 := "AL1_8" AND "AL1_8";
   "IEC_Timer_0_DB_123".TP(IN := #_w1, PT := T#50MS);
   IF "IEC_Timer_0_DB_123".Q THEN "IO BITS".HOOTER := TRUE; END_IF;
   "IEC_Timer_0_DB_152".TON(IN := #_w1, PT := T#100MS);
END_REGION

REGION Network 23: VACUUM LEAK FAIL
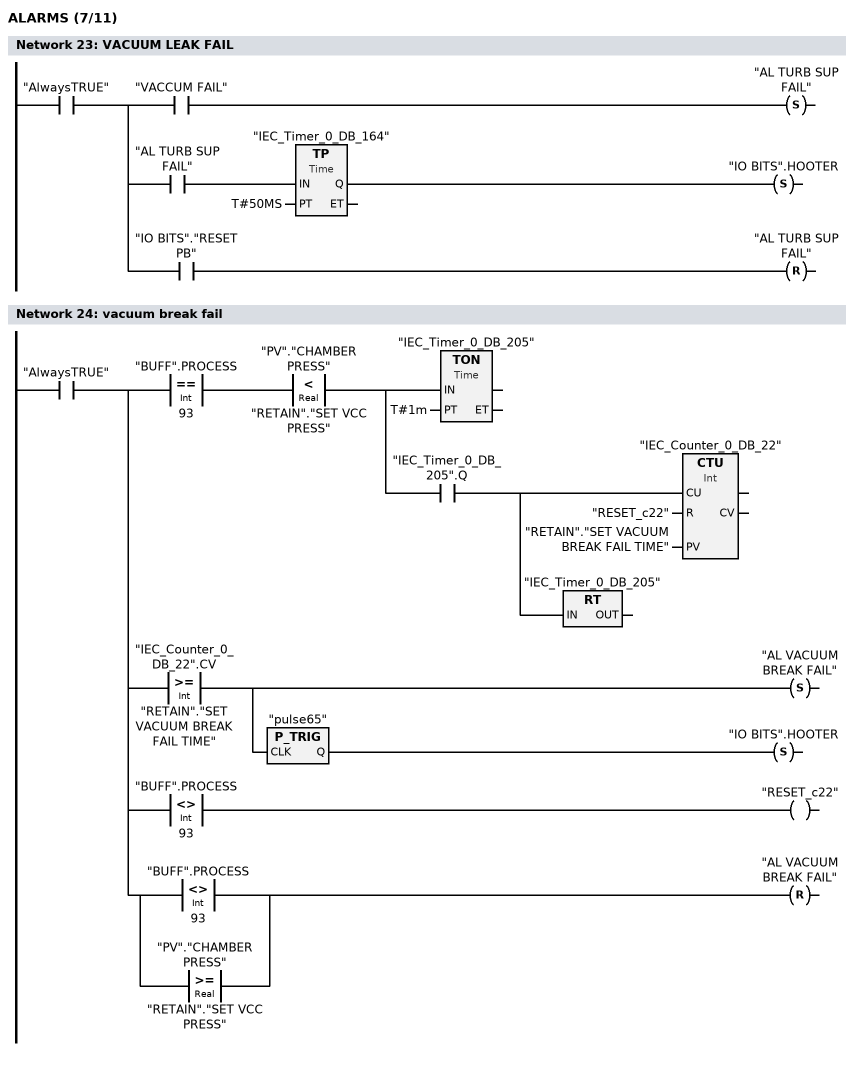
   RUNG wire#powerrail
      Contact( "AlwaysTRUE" )
      wire#w1
      Contact( "VACCUM FAIL" )
      S_Coil( "AL TURB SUP FAIL" )
   END_RUNG
   RUNG wire#w1
      Contact( "AL TURB SUP FAIL" )
      { S7_Templates := "time_type := Time" } "IEC_Timer_0_DB_164".TP(pt := T#50MS, et =>)
      S_Coil( "IO BITS".HOOTER )
   END_RUNG
   RUNG wire#w1
      Contact( "IO BITS"."RESET PB" )
      R_Coil( "AL TURB SUP FAIL" )
   END_RUNG
   // the same network as SCL:
   IF "AlwaysTRUE" AND "VACCUM FAIL" THEN "AL TURB SUP FAIL" := TRUE; END_IF;
   "IEC_Timer_0_DB_164".TP(IN := "AlwaysTRUE" AND "AL TURB SUP FAIL", PT := T#50MS);
   IF "IEC_Timer_0_DB_164".Q THEN "IO BITS".HOOTER := TRUE; END_IF;
   IF "AlwaysTRUE" AND "IO BITS"."RESET PB" THEN "AL TURB SUP FAIL" := FALSE; END_IF;
END_REGION

REGION Network 24: vacuum break fail
   RUNG wire#powerrail
      Contact( "AlwaysTRUE" )
      wire#w1
      { S7_Templates := "SrcType := Int" } EQ_Contact(in1 := "BUFF".PROCESS, in2 := 93)
      { S7_Templates := "SrcType := Real" } LT_Contact(in1 := "PV"."CHAMBER PRESS", in2 := "RETAIN"."SET VCC PRESS")
      wire#w2
      { S7_Templates := "time_type := Time" } "IEC_Timer_0_DB_205".TON(pt := T#1m, et =>)
   END_RUNG
   RUNG wire#w2
      Contact( "IEC_Timer_0_DB_205".Q )
      wire#w3
      { S7_Templates := "value_type := Int" } "IEC_Counter_0_DB_22".CTU(r := "RESET_c22", pv := "RETAIN"."SET VACUUM BREAK FAIL TIME", cv =>)
   END_RUNG
   RUNG wire#w3
      RT_Coil( "IEC_Timer_0_DB_205" )
   END_RUNG
   RUNG wire#w1
      { S7_Templates := "SrcType := Int" } GE_Contact(in1 := "IEC_Counter_0_DB_22".CV, in2 := "RETAIN"."SET VACUUM BREAK FAIL TIME")
      wire#w4
      S_Coil( "AL VACUUM BREAK FAIL" )
   END_RUNG
   RUNG wire#w4
      P_Trig( "pulse65" )
      S_Coil( "IO BITS".HOOTER )
   END_RUNG
   RUNG wire#w1
      { S7_Templates := "SrcType := Int" } NE_Contact(in1 := "BUFF".PROCESS, in2 := 93)
      Coil( "RESET_c22" )
   END_RUNG
   RUNG wire#w1
      { S7_Templates := "SrcType := Int" } NE_Contact(in1 := "BUFF".PROCESS, in2 := 93)
      wire#w5
      R_Coil( "AL VACUUM BREAK FAIL" )
   END_RUNG
   RUNG wire#w1
      { S7_Templates := "SrcType := Real" } GE_Contact(in1 := "PV"."CHAMBER PRESS", in2 := "RETAIN"."SET VCC PRESS")
   END_RUNG wire#w5
   // the same network as SCL:
   #_w1 := "AlwaysTRUE" AND ("BUFF".PROCESS = 93) AND ("PV"."CHAMBER PRESS" < "RETAIN"."SET VCC PRESS");
   "IEC_Timer_0_DB_205".TON(IN := #_w1, PT := T#1m);
   #_w2 := #_w1 AND "IEC_Timer_0_DB_205".Q;
   "IEC_Counter_0_DB_22".CTU(CU := #_w2, R := "RESET_c22", PV := "RETAIN"."SET VACUUM BREAK FAIL TIME");
   IF #_w2 THEN RESET_TIMER("IEC_Timer_0_DB_205"); END_IF;
   #_w3 := "AlwaysTRUE" AND ("IEC_Counter_0_DB_22".CV >= "RETAIN"."SET VACUUM BREAK FAIL TIME");
   IF #_w3 THEN "AL VACUUM BREAK FAIL" := TRUE; END_IF;
   #_w4 := #_w3 AND NOT "pulse65";   // rising edge
   "pulse65" := #_w3;
   IF #_w4 THEN "IO BITS".HOOTER := TRUE; END_IF;
   "RESET_c22" := "AlwaysTRUE" AND ("BUFF".PROCESS <> 93);
   IF "AlwaysTRUE" AND (("BUFF".PROCESS <> 93) OR ("PV"."CHAMBER PRESS" >= "RETAIN"."SET VCC PRESS")) THEN
       "AL VACUUM BREAK FAIL" := FALSE;
   END_IF;
END_REGION

REGION Network 25: JACKET ALARM TIME
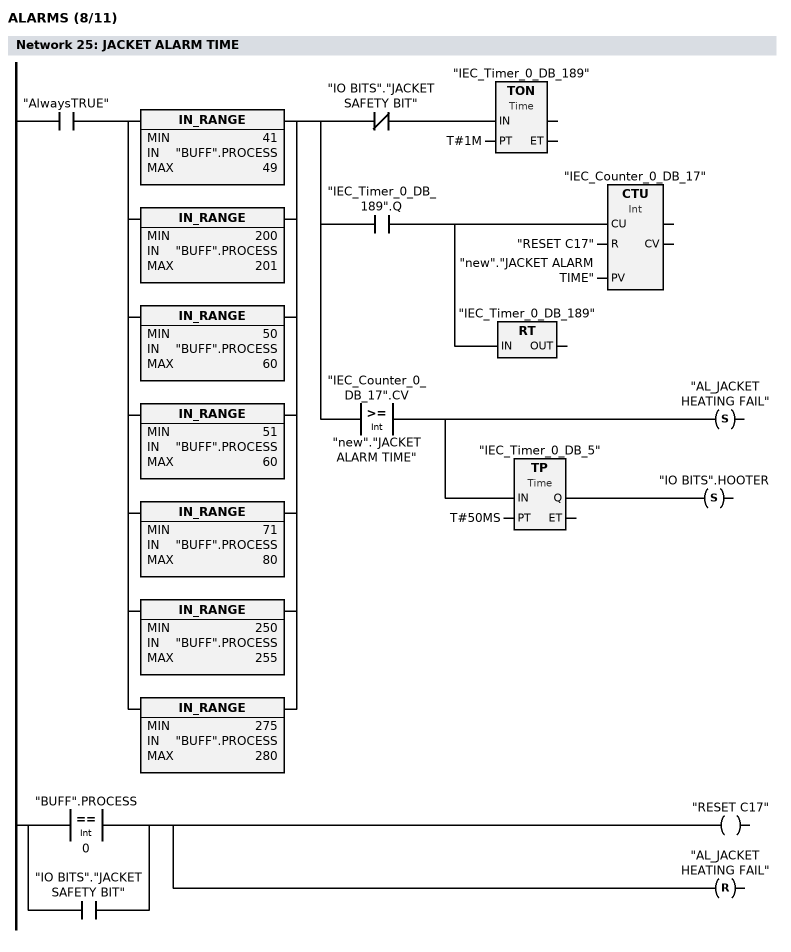
   RUNG wire#powerrail
      Contact( "AlwaysTRUE" )
      wire#w1
      { S7_Templates := "SrcType := Int" } InRange(min := 41, in := "BUFF".PROCESS, max := 49)
      wire#w2
      I_Contact( "IO BITS"."JACKET SAFETY BIT" )
      { S7_Templates := "time_type := Time" } "IEC_Timer_0_DB_189".TON(pt := T#1M, et =>)
   END_RUNG
   RUNG wire#w1
      { S7_Templates := "SrcType := Int" } InRange(min := 200, in := "BUFF".PROCESS, max := 201)
   END_RUNG wire#w2
   RUNG wire#w1
      { S7_Templates := "SrcType := Int" } InRange(min := 50, in := "BUFF".PROCESS, max := 60)
   END_RUNG wire#w2
   RUNG wire#w1
      { S7_Templates := "SrcType := Int" } InRange(min := 51, in := "BUFF".PROCESS, max := 60)
   END_RUNG wire#w2
   RUNG wire#w1
      { S7_Templates := "SrcType := Int" } InRange(min := 71, in := "BUFF".PROCESS, max := 80)
   END_RUNG wire#w2
   RUNG wire#w1
      { S7_Templates := "SrcType := Int" } InRange(min := 250, in := "BUFF".PROCESS, max := 255)
   END_RUNG wire#w2
   RUNG wire#w1
      { S7_Templates := "SrcType := Int" } InRange(min := 275, in := "BUFF".PROCESS, max := 280)
   END_RUNG wire#w2
   RUNG wire#w2
      Contact( "IEC_Timer_0_DB_189".Q )
      wire#w3
      { S7_Templates := "value_type := Int" } "IEC_Counter_0_DB_17".CTU(r := "RESET C17", pv := "new"."JACKET ALARM TIME", cv =>)
   END_RUNG
   RUNG wire#w3
      RT_Coil( "IEC_Timer_0_DB_189" )
   END_RUNG
   RUNG wire#w2
      { S7_Templates := "SrcType := Int" } GE_Contact(in1 := "IEC_Counter_0_DB_17".CV, in2 := "new"."JACKET ALARM TIME")
      wire#w4
      S_Coil( "AL_JACKET HEATING FAIL" )
   END_RUNG
   RUNG wire#w4
      { S7_Templates := "time_type := Time" } "IEC_Timer_0_DB_5".TP(pt := T#50MS, et =>)
      S_Coil( "IO BITS".HOOTER )
   END_RUNG
   RUNG wire#powerrail
      { S7_Templates := "SrcType := Int" } EQ_Contact(in1 := "BUFF".PROCESS, in2 := 0)
      wire#w5
      Coil( "RESET C17" )
   END_RUNG
   RUNG wire#powerrail
      Contact( "IO BITS"."JACKET SAFETY BIT" )
   END_RUNG wire#w5
   RUNG wire#w5
      R_Coil( "AL_JACKET HEATING FAIL" )
   END_RUNG
   // the same network as SCL:
   #_w1 := "AlwaysTRUE" AND (((41 <= "BUFF".PROCESS) AND ("BUFF".PROCESS <= 49)) OR ((200 <= "BUFF".PROCESS) AND ("BUFF".PROCESS <= 201)) OR ((50 <= "BUFF".PROCESS) AND ("BUFF".PROCESS <= 60)) OR ((51 <= "BUFF".PROCESS) AND ("BUFF".PROCESS <= 60)) OR ((71 <= "BUFF".PROCESS) AND ("BUFF".PROCESS <= 80)) OR ((250 <= "BUFF".PROCESS) AND ("BUFF".PROCESS <= 255)) OR ((275 <= "BUFF".PROCESS) AND ("BUFF".PROCESS <= 280)));
   "IEC_Timer_0_DB_189".TON(IN := #_w1 AND NOT "IO BITS"."JACKET SAFETY BIT", PT := T#1M);
   #_w2 := #_w1 AND "IEC_Timer_0_DB_189".Q;
   "IEC_Counter_0_DB_17".CTU(CU := #_w2, R := "RESET C17", PV := "new"."JACKET ALARM TIME");
   IF #_w2 THEN RESET_TIMER("IEC_Timer_0_DB_189"); END_IF;
   #_w3 := #_w1 AND ("IEC_Counter_0_DB_17".CV >= "new"."JACKET ALARM TIME");
   IF #_w3 THEN "AL_JACKET HEATING FAIL" := TRUE; END_IF;
   "IEC_Timer_0_DB_5".TP(IN := #_w3, PT := T#50MS);
   IF "IEC_Timer_0_DB_5".Q THEN "IO BITS".HOOTER := TRUE; END_IF;
   "RESET C17" := ("BUFF".PROCESS = 0) OR "IO BITS"."JACKET SAFETY BIT";
   IF "RESET C17" THEN "AL_JACKET HEATING FAIL" := FALSE; END_IF;
END_REGION

REGION Network 26: heatup ALARM TIME
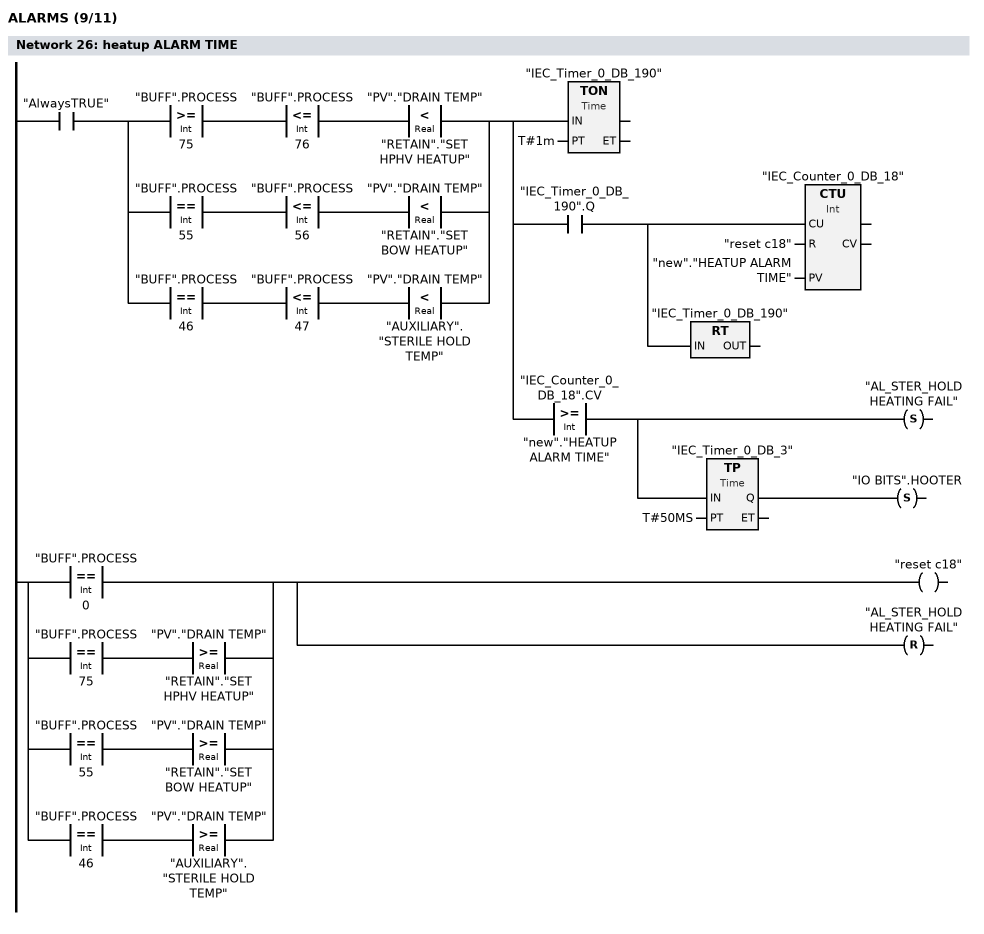
   RUNG wire#powerrail
      Contact( "AlwaysTRUE" )
      wire#w1
      { S7_Templates := "SrcType := Int" } GE_Contact(in1 := "BUFF".PROCESS, in2 := 75)
      { S7_Templates := "SrcType := Int" } LE_Contact(in1 := "BUFF".PROCESS, in2 := 76)
      { S7_Templates := "SrcType := Real" } LT_Contact(in1 := "PV"."DRAIN TEMP", in2 := "RETAIN"."SET HPHV HEATUP")
      wire#w2
      { S7_Templates := "time_type := Time" } "IEC_Timer_0_DB_190".TON(pt := T#1m, et =>)
   END_RUNG
   RUNG wire#w1
      { S7_Templates := "SrcType := Int" } EQ_Contact(in1 := "BUFF".PROCESS, in2 := 55)
      { S7_Templates := "SrcType := Int" } LE_Contact(in1 := "BUFF".PROCESS, in2 := 56)
      { S7_Templates := "SrcType := Real" } LT_Contact(in1 := "PV"."DRAIN TEMP", in2 := "RETAIN"."SET BOW HEATUP")
   END_RUNG wire#w2
   RUNG wire#w1
      { S7_Templates := "SrcType := Int" } EQ_Contact(in1 := "BUFF".PROCESS, in2 := 46)
      { S7_Templates := "SrcType := Int" } LE_Contact(in1 := "BUFF".PROCESS, in2 := 47)
      { S7_Templates := "SrcType := Real" } LT_Contact(in1 := "PV"."DRAIN TEMP", in2 := "AUXILIARY"."STERILE HOLD TEMP")
   END_RUNG wire#w2
   RUNG wire#w2
      Contact( "IEC_Timer_0_DB_190".Q )
      wire#w3
      { S7_Templates := "value_type := Int" } "IEC_Counter_0_DB_18".CTU(r := "reset c18", pv := "new"."HEATUP ALARM TIME", cv =>)
   END_RUNG
   RUNG wire#w3
      RT_Coil( "IEC_Timer_0_DB_190" )
   END_RUNG
   RUNG wire#w2
      { S7_Templates := "SrcType := Int" } GE_Contact(in1 := "IEC_Counter_0_DB_18".CV, in2 := "new"."HEATUP ALARM TIME")
      wire#w4
      S_Coil( "AL_STER_HOLD HEATING FAIL" )
   END_RUNG
   RUNG wire#w4
      { S7_Templates := "time_type := Time" } "IEC_Timer_0_DB_3".TP(pt := T#50MS, et =>)
      S_Coil( "IO BITS".HOOTER )
   END_RUNG
   RUNG wire#powerrail
      { S7_Templates := "SrcType := Int" } EQ_Contact(in1 := "BUFF".PROCESS, in2 := 0)
      wire#w5
      Coil( "reset c18" )
   END_RUNG
   RUNG wire#powerrail
      { S7_Templates := "SrcType := Int" } EQ_Contact(in1 := "BUFF".PROCESS, in2 := 75)
      { S7_Templates := "SrcType := Real" } GE_Contact(in1 := "PV"."DRAIN TEMP", in2 := "RETAIN"."SET HPHV HEATUP")
   END_RUNG wire#w5
   RUNG wire#powerrail
      { S7_Templates := "SrcType := Int" } EQ_Contact(in1 := "BUFF".PROCESS, in2 := 55)
      { S7_Templates := "SrcType := Real" } GE_Contact(in1 := "PV"."DRAIN TEMP", in2 := "RETAIN"."SET BOW HEATUP")
   END_RUNG wire#w5
   RUNG wire#powerrail
      { S7_Templates := "SrcType := Int" } EQ_Contact(in1 := "BUFF".PROCESS, in2 := 46)
      { S7_Templates := "SrcType := Real" } GE_Contact(in1 := "PV"."DRAIN TEMP", in2 := "AUXILIARY"."STERILE HOLD TEMP")
   END_RUNG wire#w5
   RUNG wire#w5
      R_Coil( "AL_STER_HOLD HEATING FAIL" )
   END_RUNG
   // the same network as SCL:
   #_w1 := "AlwaysTRUE" AND ((("BUFF".PROCESS >= 75) AND ("BUFF".PROCESS <= 76) AND ("PV"."DRAIN TEMP" < "RETAIN"."SET HPHV HEATUP")) OR (("BUFF".PROCESS = 55) AND ("BUFF".PROCESS <= 56) AND ("PV"."DRAIN TEMP" < "RETAIN"."SET BOW HEATUP")) OR (("BUFF".PROCESS = 46) AND ("BUFF".PROCESS <= 47) AND ("PV"."DRAIN TEMP" < "AUXILIARY"."STERILE HOLD TEMP")));
   "IEC_Timer_0_DB_190".TON(IN := #_w1, PT := T#1m);
   #_w2 := #_w1 AND "IEC_Timer_0_DB_190".Q;
   "IEC_Counter_0_DB_18".CTU(CU := #_w2, R := "reset c18", PV := "new"."HEATUP ALARM TIME");
   IF #_w2 THEN RESET_TIMER("IEC_Timer_0_DB_190"); END_IF;
   #_w3 := #_w1 AND ("IEC_Counter_0_DB_18".CV >= "new"."HEATUP ALARM TIME");
   IF #_w3 THEN "AL_STER_HOLD HEATING FAIL" := TRUE; END_IF;
   "IEC_Timer_0_DB_3".TP(IN := #_w3, PT := T#50MS);
   IF "IEC_Timer_0_DB_3".Q THEN "IO BITS".HOOTER := TRUE; END_IF;
   "reset c18" := ("BUFF".PROCESS = 0) OR (("BUFF".PROCESS = 75) AND ("PV"."DRAIN TEMP" >= "RETAIN"."SET HPHV HEATUP")) OR (("BUFF".PROCESS = 55) AND ("PV"."DRAIN TEMP" >= "RETAIN"."SET BOW HEATUP")) OR (("BUFF".PROCESS = 46) AND ("PV"."DRAIN TEMP" >= "AUXILIARY"."STERILE HOLD TEMP"));
   IF "reset c18" THEN "AL_STER_HOLD HEATING FAIL" := FALSE; END_IF;
END_REGION

REGION Network 27: VACUUM NOT AVAILABLE
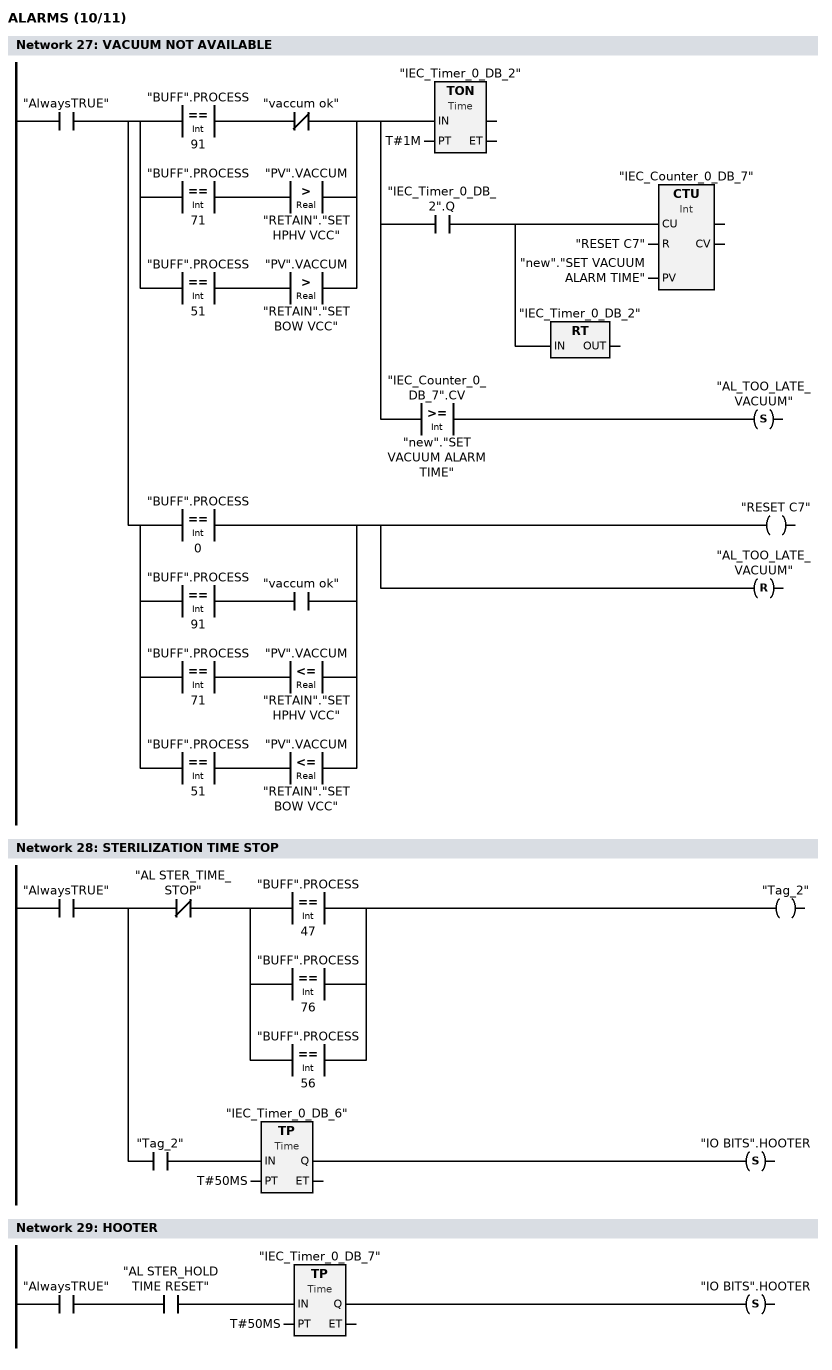
   RUNG wire#powerrail
      Contact( "AlwaysTRUE" )
      wire#w1
      { S7_Templates := "SrcType := Int" } EQ_Contact(in1 := "BUFF".PROCESS, in2 := 91)
      I_Contact( "vaccum ok" )
      wire#w2
      { S7_Templates := "time_type := Time" } "IEC_Timer_0_DB_2".TON(pt := T#1M, et =>)
   END_RUNG
   RUNG wire#w1
      { S7_Templates := "SrcType := Int" } EQ_Contact(in1 := "BUFF".PROCESS, in2 := 71)
      { S7_Templates := "SrcType := Real" } GT_Contact(in1 := "PV".VACCUM, in2 := "RETAIN"."SET HPHV VCC")
   END_RUNG wire#w2
   RUNG wire#w1
      { S7_Templates := "SrcType := Int" } EQ_Contact(in1 := "BUFF".PROCESS, in2 := 51)
      { S7_Templates := "SrcType := Real" } GT_Contact(in1 := "PV".VACCUM, in2 := "RETAIN"."SET BOW VCC")
   END_RUNG wire#w2
   RUNG wire#w2
      Contact( "IEC_Timer_0_DB_2".Q )
      wire#w3
      { S7_Templates := "value_type := Int" } "IEC_Counter_0_DB_7".CTU(r := "RESET C7", pv := "new"."SET VACUUM ALARM TIME", cv =>)
   END_RUNG
   RUNG wire#w3
      RT_Coil( "IEC_Timer_0_DB_2" )
   END_RUNG
   RUNG wire#w2
      { S7_Templates := "SrcType := Int" } GE_Contact(in1 := "IEC_Counter_0_DB_7".CV, in2 := "new"."SET VACUUM ALARM TIME")
      S_Coil( "AL_TOO_LATE_VACUUM" )
   END_RUNG
   RUNG wire#w1
      { S7_Templates := "SrcType := Int" } EQ_Contact(in1 := "BUFF".PROCESS, in2 := 0)
      wire#w4
      Coil( "RESET C7" )
   END_RUNG
   RUNG wire#w1
      { S7_Templates := "SrcType := Int" } EQ_Contact(in1 := "BUFF".PROCESS, in2 := 91)
      Contact( "vaccum ok" )
   END_RUNG wire#w4
   RUNG wire#w1
      { S7_Templates := "SrcType := Int" } EQ_Contact(in1 := "BUFF".PROCESS, in2 := 71)
      { S7_Templates := "SrcType := Real" } LE_Contact(in1 := "PV".VACCUM, in2 := "RETAIN"."SET HPHV VCC")
   END_RUNG wire#w4
   RUNG wire#w1
      { S7_Templates := "SrcType := Int" } EQ_Contact(in1 := "BUFF".PROCESS, in2 := 51)
      { S7_Templates := "SrcType := Real" } LE_Contact(in1 := "PV".VACCUM, in2 := "RETAIN"."SET BOW VCC")
   END_RUNG wire#w4
   RUNG wire#w4
      R_Coil( "AL_TOO_LATE_VACUUM" )
   END_RUNG
   // the same network as SCL:
   #_w1 := "AlwaysTRUE" AND ((("BUFF".PROCESS = 91) AND NOT "vaccum ok") OR (("BUFF".PROCESS = 71) AND ("PV".VACCUM > "RETAIN"."SET HPHV VCC")) OR (("BUFF".PROCESS = 51) AND ("PV".VACCUM > "RETAIN"."SET BOW VCC")));
   "IEC_Timer_0_DB_2".TON(IN := #_w1, PT := T#1M);
   #_w2 := #_w1 AND "IEC_Timer_0_DB_2".Q;
   "IEC_Counter_0_DB_7".CTU(CU := #_w2, R := "RESET C7", PV := "new"."SET VACUUM ALARM TIME");
   IF #_w2 THEN RESET_TIMER("IEC_Timer_0_DB_2"); END_IF;
   IF #_w1 AND ("IEC_Counter_0_DB_7".CV >= "new"."SET VACUUM ALARM TIME") THEN
       "AL_TOO_LATE_VACUUM" := TRUE;
   END_IF;
   "RESET C7" := "AlwaysTRUE" AND (("BUFF".PROCESS = 0) OR (("BUFF".PROCESS = 91) AND "vaccum ok") OR (("BUFF".PROCESS = 71) AND ("PV".VACCUM <= "RETAIN"."SET HPHV VCC")) OR (("BUFF".PROCESS = 51) AND ("PV".VACCUM <= "RETAIN"."SET BOW VCC")));
   IF "RESET C7" THEN "AL_TOO_LATE_VACUUM" := FALSE; END_IF;
END_REGION

REGION Network 28: STERILIZATION TIME STOP
   RUNG wire#powerrail
      Contact( "AlwaysTRUE" )
      wire#w1
      I_Contact( "AL STER_TIME_STOP" )
      wire#w2
      { S7_Templates := "SrcType := Int" } EQ_Contact(in1 := "BUFF".PROCESS, in2 := 47)
      wire#w3
      Coil( "Tag_2" )
   END_RUNG
   RUNG wire#w2
      { S7_Templates := "SrcType := Int" } EQ_Contact(in1 := "BUFF".PROCESS, in2 := 76)
   END_RUNG wire#w3
   RUNG wire#w2
      { S7_Templates := "SrcType := Int" } EQ_Contact(in1 := "BUFF".PROCESS, in2 := 56)
   END_RUNG wire#w3
   RUNG wire#w1
      Contact( "Tag_2" )
      { S7_Templates := "time_type := Time" } "IEC_Timer_0_DB_6".TP(pt := T#50MS, et =>)
      S_Coil( "IO BITS".HOOTER )
   END_RUNG
   // the same network as SCL:
   "Tag_2" := "AlwaysTRUE" AND NOT "AL STER_TIME_STOP" AND (("BUFF".PROCESS = 47) OR ("BUFF".PROCESS = 76) OR ("BUFF".PROCESS = 56));
   "IEC_Timer_0_DB_6".TP(IN := "AlwaysTRUE" AND "Tag_2", PT := T#50MS);
   IF "IEC_Timer_0_DB_6".Q THEN "IO BITS".HOOTER := TRUE; END_IF;
END_REGION

REGION Network 29: HOOTER
   RUNG wire#powerrail
      Contact( "AlwaysTRUE" )
      Contact( "AL STER_HOLD TIME RESET" )
      { S7_Templates := "time_type := Time" } "IEC_Timer_0_DB_7".TP(pt := T#50MS, et =>)
      S_Coil( "IO BITS".HOOTER )
   END_RUNG
   // the same network as SCL:
   "IEC_Timer_0_DB_7".TP(IN := "AlwaysTRUE" AND "AL STER_HOLD TIME RESET", PT := T#50MS);
   IF "IEC_Timer_0_DB_7".Q THEN "IO BITS".HOOTER := TRUE; END_IF;
END_REGION

REGION Network 30: boiler water level low
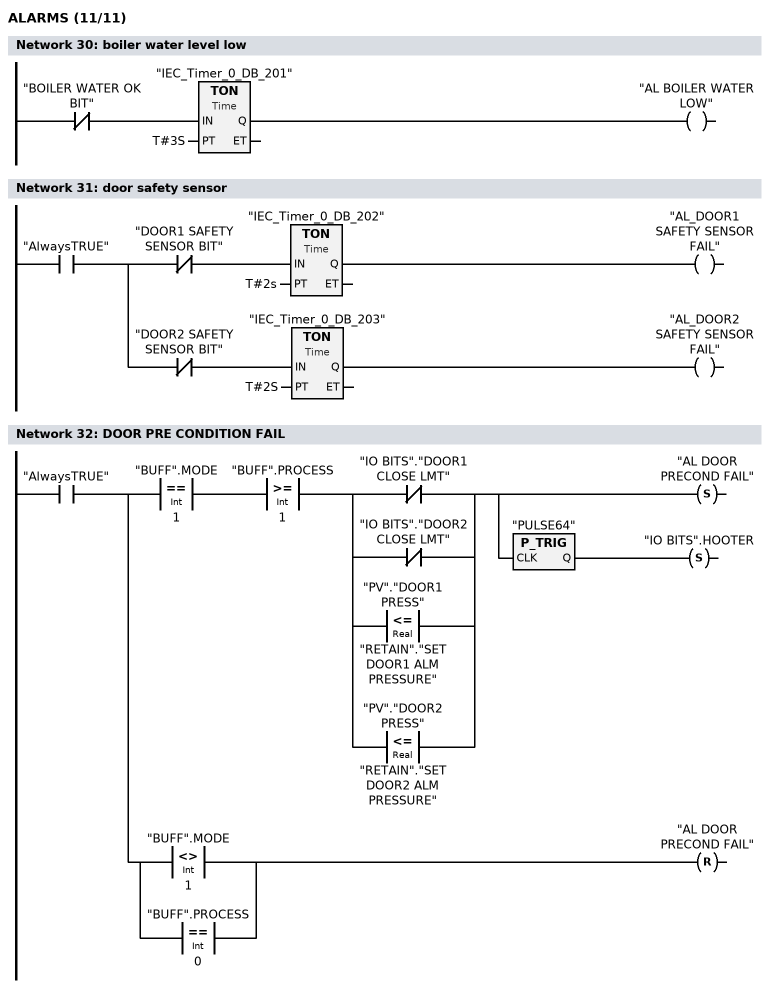
   RUNG wire#powerrail
      I_Contact( "BOILER WATER OK BIT" )
      { S7_Templates := "time_type := Time" } "IEC_Timer_0_DB_201".TON(pt := T#3S, et =>)
      Coil( "AL BOILER WATER LOW" )
   END_RUNG
   // the same network as SCL:
   "IEC_Timer_0_DB_201".TON(IN := NOT "BOILER WATER OK BIT", PT := T#3S);
   "AL BOILER WATER LOW" := "IEC_Timer_0_DB_201".Q;
END_REGION

REGION Network 31: door safety sensor
   RUNG wire#powerrail
      Contact( "AlwaysTRUE" )
      wire#w1
      I_Contact( "DOOR1 SAFETY SENSOR BIT" )
      { S7_Templates := "time_type := Time" } "IEC_Timer_0_DB_202".TON(pt := T#2s, et =>)
      Coil( "AL_DOOR1 SAFETY SENSOR FAIL" )
   END_RUNG
   RUNG wire#w1
      I_Contact( "DOOR2 SAFETY SENSOR BIT" )
      { S7_Templates := "time_type := Time" } "IEC_Timer_0_DB_203".TON(pt := T#2S, et =>)
      Coil( "AL_DOOR2 SAFETY SENSOR FAIL" )
   END_RUNG
   // the same network as SCL:
   "IEC_Timer_0_DB_202".TON(IN := "AlwaysTRUE" AND NOT "DOOR1 SAFETY SENSOR BIT", PT := T#2s);
   "AL_DOOR1 SAFETY SENSOR FAIL" := "IEC_Timer_0_DB_202".Q;
   "IEC_Timer_0_DB_203".TON(IN := "AlwaysTRUE" AND NOT "DOOR2 SAFETY SENSOR BIT", PT := T#2S);
   "AL_DOOR2 SAFETY SENSOR FAIL" := "IEC_Timer_0_DB_203".Q;
END_REGION

REGION Network 32: DOOR PRE CONDITION FAIL
   RUNG wire#powerrail
      Contact( "AlwaysTRUE" )
      wire#w1
      { S7_Templates := "SrcType := Int" } EQ_Contact(in1 := "BUFF".MODE, in2 := 1)
      { S7_Templates := "SrcType := Int" } GE_Contact(in1 := "BUFF".PROCESS, in2 := 1)
      wire#w2
      I_Contact( "IO BITS"."DOOR1 CLOSE LMT" )
      wire#w3
      S_Coil( "AL DOOR PRECOND FAIL" )
   END_RUNG
   RUNG wire#w2
      I_Contact( "IO BITS"."DOOR2 CLOSE LMT" )
   END_RUNG wire#w3
   RUNG wire#w2
      { S7_Templates := "SrcType := Real" } LE_Contact(in1 := "PV"."DOOR1 PRESS", in2 := "RETAIN"."SET DOOR1 ALM PRESSURE")
   END_RUNG wire#w3
   RUNG wire#w2
      { S7_Templates := "SrcType := Real" } LE_Contact(in1 := "PV"."DOOR2 PRESS", in2 := "RETAIN"."SET DOOR2 ALM PRESSURE")
   END_RUNG wire#w3
   RUNG wire#w3
      P_Trig( "PULSE64" )
      S_Coil( "IO BITS".HOOTER )
   END_RUNG
   RUNG wire#w1
      { S7_Templates := "SrcType := Int" } NE_Contact(in1 := "BUFF".MODE, in2 := 1)
      wire#w4
      R_Coil( "AL DOOR PRECOND FAIL" )
   END_RUNG
   RUNG wire#w1
      { S7_Templates := "SrcType := Int" } EQ_Contact(in1 := "BUFF".PROCESS, in2 := 0)
   END_RUNG wire#w4
   // the same network as SCL:
   #_w1 := "AlwaysTRUE" AND ("BUFF".MODE = 1) AND ("BUFF".PROCESS >= 1) AND (NOT "IO BITS"."DOOR1 CLOSE LMT" OR NOT "IO BITS"."DOOR2 CLOSE LMT" OR ("PV"."DOOR1 PRESS" <= "RETAIN"."SET DOOR1 ALM PRESSURE") OR ("PV"."DOOR2 PRESS" <= "RETAIN"."SET DOOR2 ALM PRESSURE"));
   IF #_w1 THEN "AL DOOR PRECOND FAIL" := TRUE; END_IF;
   #_w2 := #_w1 AND NOT "PULSE64";   // rising edge
   "PULSE64" := #_w1;
   IF #_w2 THEN "IO BITS".HOOTER := TRUE; END_IF;
   IF "AlwaysTRUE" AND (("BUFF".MODE <> 1) OR ("BUFF".PROCESS = 0)) THEN
       "AL DOOR PRECOND FAIL" := FALSE;
   END_IF;
END_REGION
END_FUNCTION
